FUNCTION ASCF_CL_35_XOR : WORD
VAR_OUTPUT
	Out								: ASCF_UnionType;		//Result of the computation (Type: VBool)
END_VAR

VAR_IN_OUT
	Arguments						: ARRAY[0..3] OF ASCF_UnionType;	//Arguments for the function (Arguments: 2 - 4, Type: VBool)

END_VAR

VAR
	tempLoopVar						: DINT;
	tempDone						: BOOL;
	tempQC							: BYTE;
	tempResult						: BOOL;
	tempValidArgumentCount			: UINT;
	constDefaultUnionType			: ASCF_UnionType;				//Union type that holds only one of its possible data types at a time. The type can be selected via the "Typeselector". Independent of the selected type, every value has a quality code "VQC".
	constUnionTypes					: ASCF_EnumUnionTypes;			//Enumeration type of the valid values for the "Typeselector" of a "GVR_unionType"-UDT.
	constQualityCodes				: ASCF_QualityCodes;				//This enum encodes the defines quality codes for the MTP standard. The values are shown in HEX. The lowest value (1) has the highest priority.    | QC Name              | Value | Priority ||----------------------|:-----:|:--------:|| Failure              | 16#00 |    1     || Function Check       | 16#60 |    2     || Ma: INTenance Request  | 16#A4 |    3     || Out of Specification | 16#68 |    4     || OK                   | 16#80 |    5     || Out of Service       | 16#1C |    6     || No Status            | 16#FF |    7     |
	constErrors						: ASCF_CL_EnumErrors;				//Enumeration type of the error codes of the Adaptive Logic.
END_VAR

VAR CONSTANT
	MIN_ARGUMENTS_COUNT				: UINT				:= 2;
END_VAR



//#################################################################################################
{region "INITIALIZE VARIABLES"}
    // #tempResult := FALSE;
    tempQC := constQualityCodes.No_Status;
    Out := constDefaultUnionType;
{endregion}

//#################################################################################################
{region "PROCESS ARGUMENTS"}
    FOR tempLoopVar := 0 TO 3 DO
        
        //-------------------------------------------------------------------------------------
        // no type --> exit loop, argument processing is done
        IF Arguments[tempLoopVar].Typeselector = constUnionTypes.None THEN
            
            tempDone := TRUE;
            
            //-------------------------------------------------------------------------------------
            // VBool --> process
        ELSIF Arguments[tempLoopVar].Typeselector = constUnionTypes.VBool THEN
            
            tempResult := tempResult XOR Arguments[tempLoopVar].VBool;
            tempQC := ASCF_CalcWQC(QC1 := tempQC, QC2 := Arguments[tempLoopVar].VQC);
            tempValidArgumentCount := tempValidArgumentCount + 1;
            
            //-------------------------------------------------------------------------------------
            // invalid type --> error
        ELSE
            ASCF_CL_35_XOR := constErrors.InvalidType;
            RETURN;
            
        END_IF;
        
        // argument processing is done --> exit loop
        IF tempDone THEN
            EXIT;
        END_IF;
        
    END_FOR;
    
    //+++++++++++++++++++++++++++++++++++++++++++++++++++++++++++++++++++++++++++++++++++++++++++++
    // too few arguments
    IF tempValidArgumentCount < MIN_ARGUMENTS_COUNT THEN
        ASCF_CL_35_XOR := constErrors.TooFewArguments;
        RETURN;
    END_IF;
{endregion}

//#################################################################################################
{region "OUTPUT"}
    Out.Typeselector := constUnionTypes.VBool;
    Out.VQC := tempQC;
    Out.VBool := tempResult;
    
    ASCF_CL_35_XOR := constErrors.None;
{endregion}

END_FUNCTION

(* stored: Version 1.1.0.1, ProductVersion 3.1.4026.4
   POU ASCF_CL_35_XOR: Id {3095d21c-ae9d-4f49-84f6-07fe035c1413}, SpecialFunc None *)
